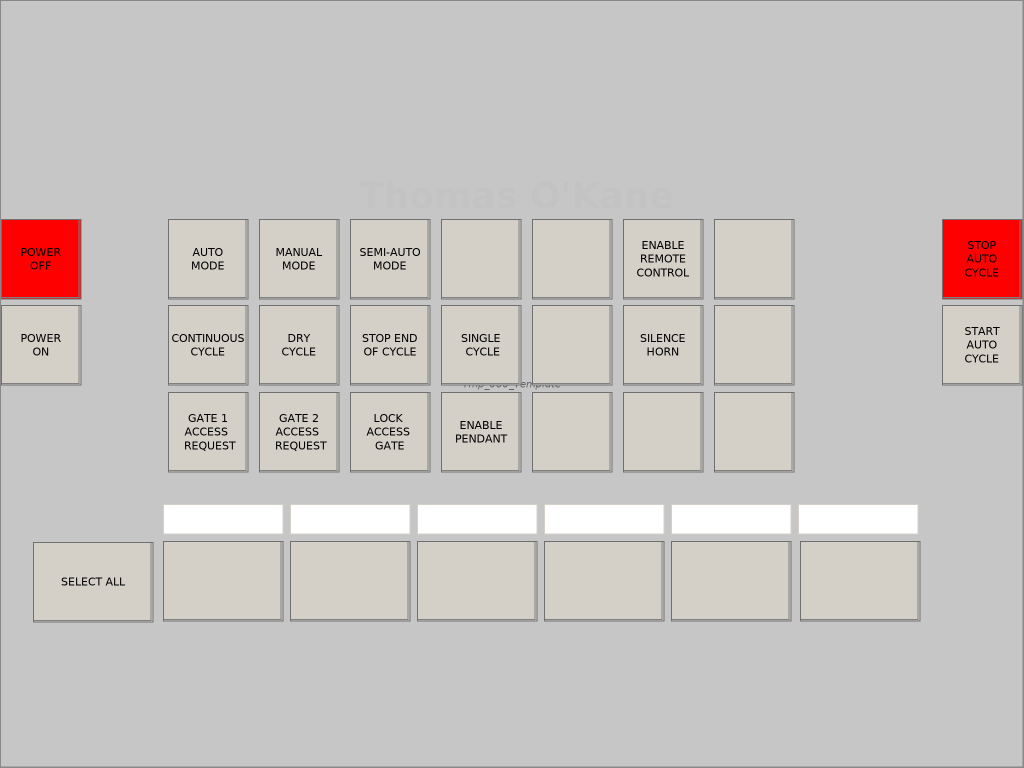
VISUALIZATION Mod_001_ModeScreen  // 1024x768
    Frame (0,0 1024x768)
        shows Tmp_000_Template(header := gHMIData.hmiHeader)
    Group (1,219 1021x166)
        Group (941,0 80x166)
            Button (0,0 80x80), "STOP AUTO CYCLE", text list: ''
                tap gHMIButtons.btnMode.btnAutoCycleStopPressed
            Button (0,86 80x80), "START AUTO CYCLE", colour toggle: gHMIButtons.btnFdbk.btnAutoCyclingFdbk, text list: ''
                tap gHMIButtons.btnMode.btnAutoCycleStartPressed
        Button (0,86 80x80), "POWER ON", colour toggle: Mc_Global.PowerOnFdbk, text list: ''
            tap gHMIButtons.btnMode.btnPowerOnPressed
        Button (0,0 80x80), "POWER OFF", text list: ''
            tap gHMIButtons.btnMode.btnPowerOffPressed
    Group (17,162 1000x310)
        Rectangle (0,0 1000x67), "Thomas O'Kane"
        Button (151,57 80x80), "AUTO MODE", colour toggle: gHMIButtons.btnFdbk.btn00Fdbk, invisible if: gHMIButtons.btnHides.btn00Hide, text list: ''
            tap gHMIButtons.btnMode.btn00Pressed
        Button (242,57 80x80), "MANUAL MODE", colour toggle: gHMIButtons.btnFdbk.btn01Fdbk, invisible if: gHMIButtons.btnHides.btn01Hide, text list: ''
            tap gHMIButtons.btnMode.btn01Pressed
        Button (333,57 80x80), "SEMI-AUTO MODE", colour toggle: gHMIButtons.btnFdbk.btn02Fdbk, invisible if: gHMIButtons.btnHides.btn02Hide, text list: ''
            tap gHMIButtons.btnMode.btn02Pressed
        Button (424,57 80x80), colour toggle: gHMIButtons.btnFdbk.btn03Fdbk, invisible if: gHMIButtons.btnHides.btn03Hide, text list: ''
            tap gHMIButtons.btnMode.btn03Pressed
        Button (606,57 80x80), "ENABLE REMOTE CONTROL", colour toggle: gHMIButtons.btnFdbk.btn05Fdbk, invisible if: gHMIButtons.btnHides.btn05Hide, text list: ''
            tap gHMIButtons.btnMode.btn05Pressed
        Button (515,57 80x80), colour toggle: gHMIButtons.btnFdbk.btn04Fdbk, invisible if: gHMIButtons.btnHides.btn04Hide, text list: ''
            tap gHMIButtons.btnMode.btn04Pressed
        Button (151,143 80x80), "CONTINUOUS CYCLE", colour toggle: gHMIButtons.btnFdbk.btn10Fdbk, invisible if: gHMIButtons.btnHides.btn10Hide, text list: ''
            tap gHMIButtons.btnMode.btn10Pressed
        Button (242,143 80x80), "DRY CYCLE", colour toggle: gHMIButtons.btnFdbk.btn11Fdbk, invisible if: gHMIButtons.btnHides.btn11Hide, text list: ''
            tap gHMIButtons.btnMode.btn11Pressed
        Button (333,143 80x80), "STOP END OF CYCLE", colour toggle: gHMIButtons.btnFdbk.btn12Fdbk, invisible if: gHMIButtons.btnHides.btn12Hide, text list: ''
            tap gHMIButtons.btnMode.btn12Pressed
        Button (424,143 80x80), "SINGLE CYCLE", colour toggle: gHMIButtons.btnFdbk.btn13Fdbk, invisible if: gHMIButtons.btnHides.btn13Hide, text list: ''
            tap gHMIButtons.btnMode.btn13Pressed
        Button (606,143 80x80), "SILENCE HORN", colour toggle: gHMIButtons.btnFdbk.btn15Fdbk, invisible if: gHMIButtons.btnHides.btn15Hide, text list: ''
            tap gHMIButtons.btnMode.btn15Pressed
        Button (515,143 80x80), colour toggle: gHMIButtons.btnFdbk.btn14Fdbk, invisible if: gHMIButtons.btnHides.btn14Hide, text list: ''
            tap gHMIButtons.btnMode.btn14Pressed
        Button (151,230 80x80), "GATE 1 ACCESS REQUEST", colour toggle: gHMIButtons.btnFdbk.btn20Fdbk, invisible if: gHMIButtons.btnHides.btn20Hide, text list: ''
            tap gHMIButtons.btnMode.btn20Pressed
        Button (242,230 80x80), "GATE 2 ACCESS REQUEST", colour toggle: gHMIButtons.btnFdbk.btn21Fdbk, invisible if: gHMIButtons.btnHides.btn21Hide, text list: ''
            tap gHMIButtons.btnMode.btn21Pressed
        Button (333,230 80x80), "LOCK ACCESS GATE", colour toggle: gHMIButtons.btnFdbk.btn22Fdbk, invisible if: gHMIButtons.btnHides.btn22Hide, text list: ''
            tap gHMIButtons.btnMode.btn22Pressed
        Button (424,230 80x80), "ENABLE PENDANT", colour toggle: gHMIButtons.btnFdbk.btn23Fdbk, invisible if: gHMIButtons.btnHides.btn23Hide, text list: ''
            tap gHMIButtons.btnMode.btn23Pressed
        Button (606,230 80x80), colour toggle: gHMIButtons.btnFdbk.btn25Fdbk, invisible if: gHMIButtons.btnHides.btn25Hide, text list: ''
            tap gHMIButtons.btnMode.btn25Pressed
        Button (515,230 80x80), colour toggle: gHMIButtons.btnFdbk.btn24Fdbk, invisible if: gHMIButtons.btnHides.btn24Hide, text list: ''
            tap gHMIButtons.btnMode.btn24Pressed
        Button (697,57 80x80), colour toggle: gHMIButtons.btnFdbk.btn06Fdbk, invisible if: gHMIButtons.btnHides.btn06Hide, text list: ''
            tap gHMIButtons.btnMode.btn06Pressed
        Button (697,143 80x80), colour toggle: gHMIButtons.btnFdbk.btn16Fdbk, invisible if: gHMIButtons.btnHides.btn16Hide, text list: ''
            tap gHMIButtons.btnMode.btn16Pressed
        Button (697,230 80x80), colour toggle: gHMIButtons.btnFdbk.btn26Fdbk, invisible if: gHMIButtons.btnHides.btn26Hide, text list: ''
            tap gHMIButtons.btnMode.btn26Pressed
    Group (33,504 887x118)
        Textfield (130,0 120x30), invisible if: NOT gHMIData.gStationEnabled[1], text list: 'ModeStates', text index: S1_Global.Data.StationState, colour variable: S1_Global.Data.StationStateColour
            p55702900: S1_Global.Data.StationStateTextColour
        Textfield (257,0 120x30), invisible if: NOT gHMIData.gStationEnabled[2], text list: 'ModeStates', text index: S2_Global.Data.StationState, colour variable: S2_Global.Data.StationStateColour
            p55702900: S2_Global.Data.StationStateTextColour
        Textfield (384,0 120x30), invisible if: NOT gHMIData.gStationEnabled[3], text list: 'ModeStates', text index: S3_Global.Data.StationState, colour variable: S3_Global.Data.StationStateColour
            p55702900: S3_Global.Data.StationStateTextColour
        Textfield (511,0 120x30), invisible if: NOT gHMIData.gStationEnabled[4], text list: 'ModeStates', text index: S4_Global.Data.StationState, colour variable: S4_Global.Data.StationStateColour
            p55702900: S4_Global.Data.StationStateTextColour
        Textfield (638,0 120x30), invisible if: NOT gHMIData.gStationEnabled[5], text list: 'ModeStates', text index: S5_Global.Data.StationState, colour variable: S5_Global.Data.StationStateColour
            p55702900: S5_Global.Data.StationStateTextColour
        Textfield (765,0 120x30), invisible if: NOT gHMIData.gStationEnabled[6], text list: 'ModeStates', text index: S6_Global.Data.StationState, colour variable: S6_Global.Data.StationStateColour
            p55702900: S6_Global.Data.StationStateTextColour
        Button (130,37 120x80), colour toggle: gHMIData.gStationSelected[1], invisible if: NOT gHMIData.gStationEnabled[1], text list: 'StationNames', text index: 1
            tap gHMIButtons.btnSelectStation1
        Button (257,37 120x80), colour toggle: gHMIData.gStationSelected[2], invisible if: NOT gHMIData.gStationEnabled[2], text list: 'StationNames', text index: 2
            tap gHMIButtons.btnSelectStation2
        Button (384,37 120x80), colour toggle: gHMIData.gStationSelected[3], invisible if: NOT gHMIData.gStationEnabled[3], text list: 'StationNames', text index: 3
            tap gHMIButtons.btnSelectStation3
        Button (511,37 120x80), colour toggle: gHMIData.gStationSelected[4], invisible if: NOT gHMIData.gStationEnabled[4], text list: 'StationNames', text index: 4
            tap gHMIButtons.btnSelectStation4
        Button (638,37 120x80), colour toggle: gHMIData.gStationSelected[5], invisible if: NOT gHMIData.gStationEnabled[5], text list: 'StationNames', text index: 5
            tap gHMIButtons.btnSelectStation5
        Button (767,37 120x80), colour toggle: gHMIData.gStationSelected[6], invisible if: NOT gHMIData.gStationEnabled[6], text list: 'StationNames', text index: 6
            tap gHMIButtons.btnSelectStation6
        Button (0,38 120x80), "SELECT ALL", colour toggle: gHMIButtons.btnAllStationsSelected, text list: ''
            tap gHMIButtons.btnSelectAll
END_VISUALIZATION

(* stored: Version 1.1.0.1, ProductVersion 3.1.4024.12
   Visu Mod_001_ModeScreen: Id {cda03302-29a3-4ca0-90e3-acf152aa8ca5} *)
